# EPICS autosave request: softGlueApp/Db/readSoftGlueCounter_ISR_settings.req
$(P)$(Q)aSub.A
$(P)$(Q)aSub.D
$(P)$(Q)cVals.NUSE
$(P)$(Q)cVals.SCAN
$(P)$(Q)oneshot
